// TwinCAT 3 PLC project UserGuidance_PLC
// ProgramVersion: 3.1.4026.14
// libraries:
//   Tc2_Standard, * (Beckhoff Automation GmbH)
//   Tc2_System, * (Beckhoff Automation GmbH)
//   Tc3_EventLogger, * (Beckhoff Automation GmbH)
// project tree:
//   / PlcTask.TcTTO
//   POUs/ MAIN.TcPOU
// real-time tasks:
//   TASK PlcTask: cycle T#10ms, priority 20, ADS port 350

CONFIGURATION UserGuidance_PLC
    RESOURCE PLC ON TwinCAT3
        TASK PlcTask(INTERVAL := T#10ms, PRIORITY := 20);
        PROGRAM MAIN WITH PlcTask : MAIN;
    END_RESOURCE
END_CONFIGURATION

// ---- POUs/MAIN.TcPOU
PROGRAM MAIN
VAR
	bSendMessagePDF	: BOOL;
	bSendMessageMP4	: BOOL;
	
	bIsInitalized 	: BOOL;
	
	fbMessagePDF	: FB_TcMessage;	
	fbMessageMP4	: FB_TcMessage;
	
	hr 				: HRESULT;
	hrLastError 	: HRESULT;
END_VAR


// init
IF NOT bIsInitalized THEN	
	bIsInitalized := TRUE;	
	hr := fbMessagePDF.CreateEx(TC_EVENTS.TestEvents.Event_PDF, 0);
	hr := fbMessageMP4.CreateEx(TC_EVENTS.TestEvents.Event_MP4, 0);
END_IF

// send message for pdf user guidance
IF bSendMessagePDF THEN
	bSendMessagePDF := FALSE;
	hr := fbMessagePDF.Send(0);
END_IF
// send message for mp4 user guidance
IF bSendMessageMP4 THEN
	bSendMessageMP4 := FALSE;
	hr := fbMessageMP4.Send(0);
END_IF

// error feedback
IF FAILED(hr) THEN
	hrLastError := hr;
END_IF

END_PROGRAM
